FUNCTION F_Concat3_Large : STRING(StringsParams.MAX_STRING_LENGTH);
VAR_IN_OUT CONSTANT
	StringOne 	: STRING(StringsParams.MAX_STRING_LENGTH);
	StringTwo	: STRING(StringsParams.MAX_STRING_LENGTH);
	StringThree	: STRING(StringsParams.MAX_STRING_LENGTH);
END_VAR
VAR
	str : STRING(StringsParams.MAX_STRING_LENGTH);
END_VAR

str := F_ConcatLarge( StringTwo, StringThree );

F_Concat3_Large := 
	F_ConcatLarge(
		StringOne, 
		str
	);

END_FUNCTION

(* stored: Version 1.1.0.1, ProductVersion 3.1.4022.6
   POU F_Concat3_Large: Id {d074b91b-6f44-48d1-b047-26a84770af6d}, SpecialFunc None *)
